// TwinCAT 3 PLC project PLC
// ProgramVersion: 3.1.4026.19
// libraries:
//   Tc2_Standard, * (Beckhoff Automation GmbH)
//   Tc2_System, * (Beckhoff Automation GmbH)
// project tree:
//   GVLs/ GVL_Var.TcGVL
//   / PlcTask.TcTTO
//   POUs/ Alarmes.TcPOU, MAIN.TcPOU (not stored), PiscaPisca.TcPOU, Simulacao.TcPOU (not stored)

CONFIGURATION PLC
    RESOURCE PLC ON TwinCAT3
        TASK PlcTask(INTERVAL := T#10ms, PRIORITY := 20);
        PROGRAM MAIN WITH PlcTask : MAIN;
        PROGRAM Simulacao WITH PlcTask : Simulacao;
    END_RESOURCE
END_CONFIGURATION

// ---- GVLs/GVL_Var.TcGVL
{attribute 'qualified_only'}
VAR_GLOBAL
	
	// Temperatura atual
	TempAtual: REAL := 7.0;
	// Setpoint de temperatura
	TempSet: REAL := 12.0;
	// Status da porta do refrigerador
	PortaAberta: BOOL := FALSE;
	// Tempo de funcionamento do compressor
	TempoCompressor: TIME := T#15s;
	// Tempo de porta aberta
	TempoPorta: TIME := T#5s;
	// Liga e desliga o compressor
	Compressor: BOOL;
	// Sinal de controle
	Sinal: BOOL;
	// Indica se a porta está aberta
	Lampada: BOOL;
END_VAR

// ---- POUs/Alarmes.TcPOU
PROGRAM Alarmes
VAR
	T1Compressor: TON;
	T2PortaAberta: TON;
	SinalIntermitente: PiscaPisca;
END_VAR

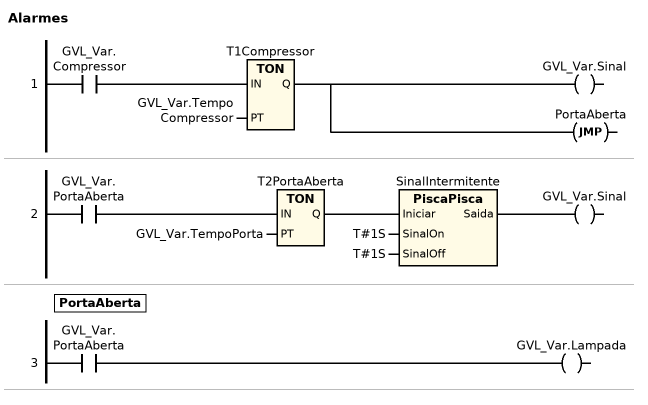
// NETWORK 1
T1Compressor(IN := GVL_Var.Compressor, PT := GVL_Var.TempoCompressor); // TON
GVL_Var.Sinal := T1Compressor.Q;
IF T1Compressor.Q THEN JMP PortaAberta; END_IF

// NETWORK 2
T2PortaAberta(IN := GVL_Var.PortaAberta, PT := GVL_Var.TempoPorta); // TON
SinalIntermitente(Iniciar := T2PortaAberta.Q, SinalOn := T#1S, SinalOff := T#1S); // PiscaPisca
GVL_Var.Sinal := SinalIntermitente.Saida;

// NETWORK 3
PortaAberta:
GVL_Var.Lampada := GVL_Var.PortaAberta;

END_PROGRAM

// ---- POUs/PiscaPisca.TcPOU
FUNCTION_BLOCK PiscaPisca
VAR_INPUT
	Iniciar: BOOL;
	SinalOn: TIME := T#1s;
	SinalOff: TIME := T#1s;
END_VAR
VAR_OUTPUT
	Saida: BOOL;
END_VAR
VAR
	T1: TON;
	T2: TON;
END_VAR

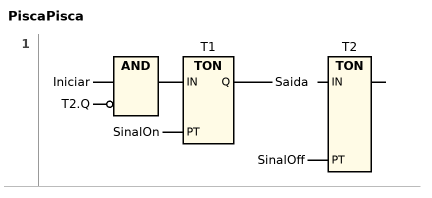
// NETWORK 1
T1(IN := Iniciar AND NOT T2.Q, PT := SinalOn); // TON
Saida := T1.Q;
T2(IN := T1.Q, PT := SinalOff); // TON

END_FUNCTION_BLOCK
